// TIA Portal V21 export
TYPE "Rcp_Generale"
TITLE = Parte Generale Della Ricetta
   STRUCT
      VelocitàMaxFormato : Word;
      Rcp_Trasporti : Int;
      "Tipo Contenitore" : Int;   // 0 = Vetro / 1 = Plastica / 2 = Lattina
   END_STRUCT;
END_TYPE
